PROGRAM MAIN
VAR
    _fbCalculator : FbCalculator;
END_VAR

END_PROGRAM

(* stored: Version 1.1.0.1, ProductVersion 3.1.4024.9
   POU MAIN: Id {267f4f9f-c3b1-4265-aa3a-a98afd343d60}, SpecialFunc None *)
